{attribute 'linkalways'} 
{attribute 'no_explicit_call' := 'This FB is a CLASS and must be accessed using methods or properties'}
{attribute 'enable_dynamic_creation'}
FUNCTION_BLOCK Node_F_VN_InsertIntoContainer_TcVnPoint2_LREAL EXTENDS VisionNode
VAR
    aElement : _TcVnPoint2_LREAL;
    ipContainer : _ITcVnContainer;
    nIndex : _ULINT(0);
    hrPrev : _HRESULT(S_OK);
    hresult : _HRESULT(S_OK);
END_VAR

METHOD PUBLIC  Clone : I_Node
VAR
	pNode : POINTER TO Node_F_VN_InsertIntoContainer_TcVnPoint2_LREAL;
END_VAR
pNode := __NEW(Node_F_VN_InsertIntoContainer_TcVnPoint2_LREAL);
Clone := pNode^;
END_METHOD

METHOD FB_init : BOOL
VAR_INPUT
	bInitRetains : BOOL; // if TRUE, the retain variables are initialized (warm start / cold start)
	bInCopyCode : BOOL;  // if TRUE, the instance afterwards gets moved into the copy code (online change)
END_VAR
AddInput('aElement', aElement);
AddInput('ipContainer', ipContainer);
AddInput('nIndex', nIndex);
AddInput('hrPrev', hrPrev);
AddOutput('ipContainer', ipContainer);
AddOutput('hresult',hresult);
END_METHOD

METHOD PROTECTED OnExecute : HRESULT
hresult.Value := F_VN_InsertIntoContainer_TcVnPoint2_LREAL(
    aElement := aElement.Value,
    ipContainer := ipContainer.Value,
    nIndex := nIndex.Value,
    hrPrev:= hrPrev.Value);
END_METHOD

METHOD PUBLIC PreExecutionCheck
VAR_INPUT
	Check : I_PreExecutionChecks;
END_VAR
Check.IsTrue(ipContainer.IsValid, 'ipContainer must be a valid container');
END_METHOD

END_FUNCTION_BLOCK

(* stored: Version 1.1.0.1, ProductVersion 3.1.4024.13
   POU Node_F_VN_InsertIntoContainer_TcVnPoint2_LREAL: Id {d35e48d1-95c9-4e9b-9619-810d8191f519}, SpecialFunc None
   Folder Constructor: Id {a327d4e5-f832-4319-b839-ae637bf64f49}
   Method Clone: Id {dd343de0-3b91-4fd2-b478-47208ca5d554}
   Method FB_init: Id {5abe4088-7b1d-4c1b-8183-ccb60c63d85a}
   Method OnExecute: Id {9625c392-9877-44ff-8ab8-968371a381cd}
   Method PreExecutionCheck: Id {3bd2cab8-9c93-4859-b3da-9eb4356190d2} *)
